(* IEC 61131-3 sources: horner-cscape-mcp/artifacts/projects/TankLevel_P5_Dedicated/pous, 3 files *)

(* ---- FB_ModbusScaleQuality.st ---- *)
FUNCTION_BLOCK FB_ModbusScaleQuality
VAR_INPUT
    RawInput : INT;
    RawMin : INT := 0;
    RawMax : INT := 32000;
    EUMin : REAL := 0.0;
    EUMax : REAL := 100.0;
    CommFailure : BOOL := FALSE;
    StaleQuality : BOOL := FALSE;
    FailSafeValue : REAL := 0.0;
END_VAR
VAR_OUTPUT
    ScaledOutput : REAL;
    QualityGood : BOOL;
    AlarmActive : BOOL;
    Underflow : BOOL;
    Overflow : BOOL;
END_VAR
VAR
    RawSpan : REAL;
    EUSpan : REAL;
    Normalized : REAL;
    CalculatedEU : REAL;
END_VAR

(* 1. Out-of-bounds Detection *)
IF RawInput < RawMin THEN
    Underflow := TRUE;
ELSE
    Underflow := FALSE;
END_IF;

IF RawInput > RawMax THEN
    Overflow := TRUE;
ELSE
    Overflow := FALSE;
END_IF;

(* 2. Communication Health & Telemetry Quality Gating *)
IF CommFailure OR StaleQuality THEN
    AlarmActive := TRUE;
    QualityGood := FALSE;
    ScaledOutput := FailSafeValue;
ELSE
    AlarmActive := FALSE;
    QualityGood := TRUE;

    (* 3. Linear Interpolation & Clamping *)
    RawSpan := INT_TO_REAL(RawMax - RawMin);
    EUSpan := EUMax - EUMin;

    IF RawSpan <> 0.0 THEN
        Normalized := INT_TO_REAL(RawInput - RawMin) / RawSpan;
        CalculatedEU := EUMin + (Normalized * EUSpan);
    ELSE
        CalculatedEU := EUMin;
    END_IF;

    IF EUMin <= EUMax THEN
        IF CalculatedEU < EUMin THEN
            ScaledOutput := EUMin;
        ELSIF CalculatedEU > EUMax THEN
            ScaledOutput := EUMax;
        ELSE
            ScaledOutput := CalculatedEU;
        END_IF;
    ELSE
        IF CalculatedEU < EUMax THEN
            ScaledOutput := EUMax;
        ELSIF CalculatedEU > EUMin THEN
            ScaledOutput := EUMin;
        ELSE
            ScaledOutput := CalculatedEU;
        END_IF;
    END_IF;
END_IF;

END_FUNCTION_BLOCK

(* ---- TankLevelControl.st ---- *)
PROGRAM TankLevelControl
VAR
    RawAnalogInput : WORD := 0; (* %AI1: Modbus Register 40001 (Wire offset 0x0000) *)
    TankLevelPV : REAL := 0.0; (* Scaled Process Variable: 0.0..100.0 % *)
    Setpoint : REAL := 50.0; (* %AQ1 *)
    AutoMode : BOOL := TRUE; (* %M1 *)
    ManualOutputCmd : REAL := 0.0; (* %AQ2 *)
    PumpCmdActive : BOOL := FALSE; (* %Q1 *)
    PumpRunningFeedback : BOOL := FALSE; (* %I1 *)
    HighAlarm : BOOL := FALSE; (* %T3 *)
    LowAlarm : BOOL := FALSE; (* %T4 *)
    ControlError : REAL := 0.0; (* %R10 *)
    HI_Limit : REAL := 75.0;
    LO_Limit : REAL := 35.0;
    CommFailureAlarm : BOOL := FALSE; (* %M10: Remote Modbus Comm Timeout Fault *)
    TankLevelPV_Stale : BOOL := FALSE; (* %M11: Stale Telemetry Quality Indicator *)
    CommWatchdogReg : WORD := 0; (* Remote Modbus Heartbeat Register *)
    LastWatchdogReg : WORD := 0;
    WatchdogTimer : TON;
END_VAR

(* 1. Modbus Communication Health & Watchdog Check *)
IF CommWatchdogReg <> LastWatchdogReg THEN
    LastWatchdogReg := CommWatchdogReg;
    CommFailureAlarm := FALSE;
    TankLevelPV_Stale := FALSE;
END_IF;

WatchdogTimer(IN := NOT CommFailureAlarm, PT := T#2s);
IF WatchdogTimer.Q THEN
    CommFailureAlarm := TRUE;
    TankLevelPV_Stale := TRUE;
END_IF;

(* 2. Modbus Telemetry Scaling & Fail-Safe Handling *)
IF NOT CommFailureAlarm THEN
    (* Linear scaling: 0.0..32000.0 count -> 0.0..100.0 % *)
    TankLevelPV := WORD_TO_REAL(RawAnalogInput) * 100.0 / 32000.0;
    TankLevelPV := LIMIT(0.0, TankLevelPV, 100.0);
ELSE
    (* Fail-safe clamp to safe state during fieldbus comm loss *)
    TankLevelPV := 0.0;
END_IF;

(* 3. Closed-Loop Tank Level Control Logic *)
ControlError := Setpoint - TankLevelPV;

IF TankLevelPV >= HI_Limit THEN
    HighAlarm := TRUE;
ELSE
    HighAlarm := FALSE;
END_IF;

IF TankLevelPV <= LO_Limit THEN
    LowAlarm := TRUE;
ELSE
    LowAlarm := FALSE;
END_IF;

IF AutoMode THEN
    IF TankLevelPV < Setpoint THEN
        PumpCmdActive := TRUE;
    ELSE
        PumpCmdActive := FALSE;
    END_IF;
ELSE
    IF ManualOutputCmd > 0.0 THEN
        PumpCmdActive := TRUE;
    ELSE
        PumpCmdActive := FALSE;
    END_IF;
END_IF;

END_PROGRAM

(* ---- TankLevelModbusBridge.st ---- *)
PROGRAM TankLevelModbusBridge
VAR
    (* Raw Modbus Telemetry Inputs *)
    AI_TankLevelRaw AT %AI1 : INT := 0;
    AI_InflowRaw AT %AI2 : INT := 0;
    AI_DischargeRaw AT %AI3 : INT := 0;

    (* Telemetry Health & Communication Flags *)
    M_LevelCommFail AT %M10 : BOOL := FALSE;
    M_LevelStale AT %M11 : BOOL := FALSE;
    M_InflowCommFail AT %M12 : BOOL := FALSE;
    M_InflowStale AT %M13 : BOOL := FALSE;
    M_DischargeCommFail AT %M14 : BOOL := FALSE;
    M_DischargeStale AT %M15 : BOOL := FALSE;

    (* Engineering Unit Scaled Process Outputs *)
    TankLevelPV AT %R101 : REAL := 0.0;
    InflowRatePV AT %R103 : REAL := 0.0;
    DischargePressPV AT %R105 : REAL := 0.0;

    (* Quality & Status Output Flags *)
    LevelQualityGood AT %M21 : BOOL := FALSE;
    LevelAlarmActive AT %M20 : BOOL := FALSE;
    LevelUnderflow AT %M26 : BOOL := FALSE;
    LevelOverflow AT %M27 : BOOL := FALSE;

    InflowQualityGood AT %M23 : BOOL := FALSE;
    InflowAlarmActive AT %M22 : BOOL := FALSE;
    InflowUnderflow AT %M28 : BOOL := FALSE;
    InflowOverflow AT %M29 : BOOL := FALSE;

    DischargeQualityGood AT %M25 : BOOL := FALSE;
    DischargeAlarmActive AT %M24 : BOOL := FALSE;
    DischargeUnderflow AT %M30 : BOOL := FALSE;
    DischargeOverflow AT %M31 : BOOL := FALSE;

    (* Function Block Instances *)
    fbLevelScale : FB_ModbusScaleQuality;
    fbInflowScale : FB_ModbusScaleQuality;
    fbDischargeScale : FB_ModbusScaleQuality;
END_VAR

(* Channel 1: Tank Level PV (0..32000 -> 0.0..100.0 %) *)
fbLevelScale(RawInput := AI_TankLevelRaw, RawMin := 0, RawMax := 32000, EUMin := 0.0, EUMax := 100.0, CommFailure := M_LevelCommFail, StaleQuality := M_LevelStale, FailSafeValue := 0.0);
TankLevelPV := fbLevelScale.ScaledOutput;
LevelQualityGood := fbLevelScale.QualityGood;
LevelAlarmActive := fbLevelScale.AlarmActive;
LevelUnderflow := fbLevelScale.Underflow;
LevelOverflow := fbLevelScale.Overflow;

(* Channel 2: Inflow Rate PV (0..32000 -> 0.0..500.0 L/min) *)
fbInflowScale(RawInput := AI_InflowRaw, RawMin := 0, RawMax := 32000, EUMin := 0.0, EUMax := 500.0, CommFailure := M_InflowCommFail, StaleQuality := M_InflowStale, FailSafeValue := 0.0);
InflowRatePV := fbInflowScale.ScaledOutput;
InflowQualityGood := fbInflowScale.QualityGood;
InflowAlarmActive := fbInflowScale.AlarmActive;
InflowUnderflow := fbInflowScale.Underflow;
InflowOverflow := fbInflowScale.Overflow;

(* Channel 3: Discharge Pressure PV (0..32000 -> 0.0..10.0 bar) *)
fbDischargeScale(RawInput := AI_DischargeRaw, RawMin := 0, RawMax := 32000, EUMin := 0.0, EUMax := 10.0, CommFailure := M_DischargeCommFail, StaleQuality := M_DischargeStale, FailSafeValue := 0.0);
DischargePressPV := fbDischargeScale.ScaledOutput;
DischargeQualityGood := fbDischargeScale.QualityGood;
DischargeAlarmActive := fbDischargeScale.AlarmActive;
DischargeUnderflow := fbDischargeScale.Underflow;
DischargeOverflow := fbDischargeScale.Overflow;

END_PROGRAM
